FUNCTION InQ : BOOL
VAR_INPUT
	iiNum: INT;
	iaQueue:ARRAY[1..3] OF INT;
END_VAR
VAR
END_VAR


IF iiNum=iaQueue[1] OR iiNum=iaQueue[2] OR iiNum=iaQueue[3] THEN
	InQueue:=TRUE;
ELSE
	InQueue:=FALSE;	
END_IF

END_FUNCTION

(* stored: Version 1.1.0.1, ProductVersion 3.1.4024.12
   POU InQ: Id {9d2c50ee-5b04-4ac3-b434-77c1e6cc5ee5}, SpecialFunc None *)
